FUNCTION_BLOCK FB_MockLight IMPLEMENTS ITrafficLight
VAR
	_state : E_LightState := E_LightState.Red;
END_VAR

{warning 'add property implementation'}
PROPERTY CurrentState : E_LightState
GET
CurrentState := _state;
END_GET
SET
_state := CurrentState;
END_SET
END_PROPERTY

END_FUNCTION_BLOCK

(* stored: Version 1.1.0.1, ProductVersion 3.1.4024.12
   POU FB_MockLight: Id {ce876cf4-4d9e-4288-9c08-708936bdc733}, SpecialFunc None
   Property CurrentState: Id {265faf78-6272-4558-8004-185fb6de5390}
   Get Get: Id {146ebe25-a190-4a6b-b422-99f5fa0b7666}
   Set Set: Id {60a51fbc-cea8-48f8-8f09-def3fa75163c} *)
